FUNCTION_BLOCK JoyStickGantryLogic
VAR_INPUT
	HookX : EtherCAT_Kid;
	HookY : EtherCAT_Kid;
	MaxTime : TIME;
	Patient : ARRAY[0..4] OF patient;
	ModeCheck : DINT;
END_VAR

VAR_IN_OUT
		sm : FB_SerialCom_Remote; //SerialRemote Assigned to Gantry
END_VAR

VAR_OUTPUT
	TrackedPatient : INT;
END_VAR

VAR
WirelessMove : WirelessMove;
X: INT;
DeadManState : BOOL;

END_VAR
////Patient1 : Patient;
//Patient2 : Patient;
//Patient3 : Patient;
//Patient4 : Patient;

IF sm.SyncPressed = 5  THEN
	GVL_HMI.GUIGlobalReset := TRUE;
	RETURN;
END_IF


IF MAIN.GlobalEstopActive THEN
	sm.ScreenCommanded := 51; 
	TrackedPatient := 0;
	RETURN;
ELSE
	IF sm.ScreenCommanded = 51 THEN sm.ScreenCommanded := 73; END_IF
END_IF


IF sm.ScreenActive =73 OR sm.ScreenActive = 74 OR sm.ScreenActive = 72 THEN
	

	sm.ScreenCommanded := 73;
	FOR X := 1 TO 4 DO
		IF ((Patient[x].X - HookX.currentPosition) * (Patient[x].X - HookX.currentPosition)) + ((Patient[x].Y - HookY.currentPosition) * (Patient[x].Y - HookY.currentPosition)) >0 THEN
			IF SQRT(((Patient[x].X - HookX.currentPosition) * (Patient[x].X - HookX.currentPosition)) + ((Patient[x].Y - HookY.currentPosition) * (Patient[x].Y - HookY.currentPosition))) < GVL_HMI.GantryLockWindow 
				AND Patient[x].AGE < T#500MS THEN
				sm.ScreenCommanded := 74;
				IF sm.ZAxisPressed > 1 AND sm.DeadmanPressed < 0 AND sm.ScreenActive = 74 THEN
					TrackedPatient := X;
					sm.ScreenCommanded := 74+ INT_TO_BYTE(X);
				END_IF
			END_IF
		END_IF
	END_FOR

END_IF

IF sm.ZAxisPressed > 2 AND sm.DeadmanPressed > 2 THEN TrackedPatient := 0; sm.ScreenCommanded := 74; END_IF

IF sm.DeadmanPressed >= 2 AND sm.ScreenActive < 75 AND sm.ScreenCommanded > 71 THEN
	ModeCheck := 1;
	WirelessMove(HookX := HookX, HookY:= HookY, sm :=SM, WindowScaling := 1);
	DeadmanState := TRUE;
ELSIF sm.DeadmanPressed < 1 AND sm.ScreenActive > 74 AND sm.ScreenCommanded > 74  AND patient[TrackedPatient].AGE < T#500MS AND sm.Age < T#1000MS THEN
		ModeCheck := 2;
	DeadmanState := TRUE;
	MAIN.Kid[Hookx.CheckIn.KidID].TargetPos := Patient[TrackedPatient].X;
	MAIN.Kid[HookY.CheckIn.KidID].TargetPos := Patient[TrackedPatient].Y;
ELSIF sm.DeadmanPressed < 0 THEN
		ModeCheck := 3;
	DeadManState := FALSE;
ELSE
		ModeCHeck := 4;

END_IF


x:= TrackedPatient;
IF TrackedPatient <> 0 THEN
	IF( Patient[x].x < -500 OR Patient[x].x > 3900 OR Patient[x].y > 9500 OR Patient[x].y < -500 OR sm.Age > T#2000MS OR Patient[x].AGE > T#500MS) THEN
		ModeCheck := ModeCheck + 10;
		sm.ScreenCommanded := 73;
		TrackedPatient := 0;
	END_IF
	if patient[x].Age > MaxTime then Maxtime := Patient[x].AGE; END_IF
END_IF



IF sm.EstopPressed > 1 THEN
	MAIN.JoyStickEstopActive := TRUE;
	
END_IF


IF HookX.CheckIn.KidID = 1 THEN
	MAIN.JoyStick1DeadMan:=DeadmanState;
ELSE
	MAIN.JoyStick2DeadMan := DeadmanState;
END_IF

END_FUNCTION_BLOCK

(* stored: Version 1.1.0.1, ProductVersion 3.1.4022.3
   POU JoyStickGantryLogic: Id {32d788c7-386b-4f66-8e8f-54d6fd322416}, SpecialFunc None *)
